PROGRAM MAIN
VAR
	test	: DINT;
END_VAR

test:=test+1;

END_PROGRAM

(* stored: Version 1.1.0.1, ProductVersion 3.1.4024.12
   POU MAIN: Id {bab0ef4a-2e3e-4ede-a8f2-ff177030bc12}, SpecialFunc None *)
